PROGRAM main
VAR
	CountPulse AT %QX0.0 : bool;
	ResetCounter AT %QX0.1 : bool;
	Done AT %QX0.2 : bool;
	PartCounter : TF_CTU;
	PartCounter_ACC AT %MD0 : dint;
END_VAR

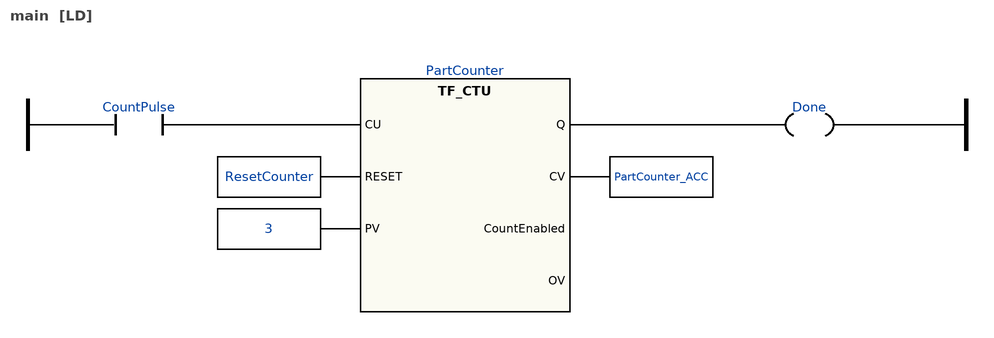
(* LD diagram, written out as Structured Text *)
PartCounter(CU := CountPulse, RESET := ResetCounter, PV := 3);
PartCounter_ACC := PartCounter.CV;
Done := PartCounter.Q;
END_PROGRAM
